TYPE ST_Joystick :
STRUCT
	X : LREAL;
	Y : LREAL;
	Topswitch : BOOL;
END_STRUCT
END_TYPE

(* stored: Version 1.1.0.1, ProductVersion 3.1.4024.12
   DUT ST_Joystick: Id {09d160ef-feca-42b6-af40-0a2998438d03} *)
